// TwinCAT 3 PLC project Simulation
// ProgramVersion: 3.1.4022.1
// libraries:
//   Tc2_Standard, * (Beckhoff Automation GmbH)
//   Tc2_System, * (Beckhoff Automation GmbH)
//   Tc3_Module, * (Beckhoff Automation GmbH)
// project tree:
//   / GlobalTextList.TcGTLO, PlcTask.TcTTO, Visualization Manager.TcVMO (not stored)
//   GVLs/ Global.TcGVL
//   GVLs/IO/ IO_Outputs.TcGVL, IO_Inputs.TcGVL
//   POUs/ FB_HeaterSimu.TcPOU, MAIN_SIMU.TcPOU
// (motion and I/O tree: see PLC project main)
// real-time tasks:
//   TASK StandardTask: cycle T#10ms, priority 1, ADS port 350
//   TASK PlcTask: cycle T#10ms, priority 20, ADS port 351
// variable links:
//   Main/Main Instance <-> Simulation/Simulation Instance
//     PlcTask Inputs/IO_Inputs.i_HtrTemp <-> PlcTask Outputs/IO_Outputs.o_HtrTemp
//     PlcTask Outputs/IO_Outputs.o_HtrON <-> PlcTask Inputs/IO_Inputs.i_HtrON
//     PlcTask Outputs/IO_Outputs.o_Restart <-> PlcTask Inputs/IO_Inputs.i_Restart

CONFIGURATION Simulation
    RESOURCE PLC ON TwinCAT3
        TASK PlcTask(INTERVAL := T#10ms, PRIORITY := 20);
        PROGRAM MAIN_SIMU WITH PlcTask : MAIN_SIMU;
    END_RESOURCE
END_CONFIGURATION

// ---- GVLs/Global.TcGVL
{attribute 'qualified_only'}
// Global simulation members
//
VAR_GLOBAL
END_VAR

// ---- GVLs/IO/IO_Outputs.TcGVL
{attribute 'qualified_only'}
// Simulated I/O Outputs
//
VAR_GLOBAL

	// Simulated output signals...
	o_HtrTemp AT %Q*: REAL; // Heater temperature [°C]
 
END_VAR

// ---- GVLs/IO/IO_Inputs.TcGVL
{attribute 'qualified_only'}
// I/O Inputs from main application
//
VAR_GLOBAL

	// Input signals from main application...
	i_HtrON   AT %I*: BOOL; // Heater to ON
	i_Restart AT %I*: BOOL; // Restart simulation

END_VAR

// ---- POUs/MAIN_SIMU.TcPOU
// Simulation application main function
//
PROGRAM MAIN_SIMU
VAR

	// Function blocks...
	fbHeaterSimu: FB_HeaterSimu; // Heater simulation

	// Other members...
	Cntr: DINT; // Counter, visiting times
	
END_VAR

// Update counter
Cntr := ( Cntr + 1 );

// Call the heater simulation
fbHeaterSimu();

END_PROGRAM

// ---- POUs/FB_HeaterSimu.TcPOU
// Simulates the heater temperature
//
FUNCTION_BLOCK FB_HeaterSimu
VAR_INPUT
END_VAR
VAR
	
	// Other members...
	Cntr:        SINT; // Counter
	Power:       SINT; // Heating power [0...100 %]
	PowerLast:   SINT; // Last heating power [0...100 %]
	Speed:       REAL; // Heating speed [+/- °C/s]
	Temperature: REAL; // Temperature [°C]
	TempTarget:  REAL; // Target temperature from the active power level [°C]
	
END_VAR

// Is restart requested ?
IF IO_Inputs.i_Restart THEN

	// Restart members
	Cntr        := 0;
	Power       := 0;
	PowerLast   := 0;
	Speed       := 0;
	Temperature := 0;
	
END_IF

// Is heater controlled to ON ?
IF IO_Inputs.i_HtrON THEN
	
	// Increase the heating power [%]
	Power := ( Power + 1 );
	
END_IF

// Is visited 100 times ?
IF Cntr = 100 THEN
	
	// Restart the visiting counter
	Cntr := 1;
	
// else, Not 100 times yet
ELSE
	
	// Increase the visiting counter
	Cntr := ( Cntr + 1 );
	RETURN;
	
END_IF

// Be sure the device movement is slow
Power := LIMIT( MAX( 0, PowerLast - 10 ), Power, MIN( 100, PowerLast + 10 ));

// Tune the power (dead time)
Power := (( Power + ( PowerLast * 2 )) / 3 );
 
// Define the final temperature based from the active power level [°C]
TempTarget := ( 10 + ( Power * 1.9 )); // 0 ...100 % => 10 ... 200 °C
  
// Define the heating speed  [+/- °C/s]
Speed := LIMIT( -2, Speed + (( TempTarget - Temperature ) / 300 ), 2 );

// Update new temperature [°C]
Temperature := LIMIT( 0, Temperature + Speed, 999 );

// Write temperature to I/O output [°C]
IO_Outputs.o_HtrTemp := Temperature;

// Save the latest power 
PowerLast := Power;
Power     := 0;

END_FUNCTION_BLOCK
